// TIA Portal V19 export
TYPE "LUC_typeMonitoring"
TITLE = LUC_typeStateModeManagerMonitoring
// Module related monitoring information
// stored: Access Published
   STRUCT
      unitModeCurrent { ExternalWritable := 'False'} : DInt;   // Current unit mode
      unitModeRequested { ExternalWritable := 'False'} : Bool;   // Requested unit mode change
      unitModeChangeInProcess { ExternalWritable := 'False'} : Bool;   // Unit mode change in process
      stateCurrent { ExternalWritable := 'False'} : DInt;   // Current state
      stateRequested { ExternalWritable := 'False'} : DInt;   // Requested state
      stateChangeInProcess { ExternalWritable := 'False'} : Bool;   // State change in process
      curDisabledStates { ExternalWritable := 'False'} : DWord;   // Disabled states in current unit mode
      curHoldCmdCfg { ExternalWritable := 'False'} : DWord;   // Bit locations within the DWORD represent State numbers. A value of 1 in a bit location indicates that the Hold control command is taken into account in the corresponding state
      curCompleteCmdCfg { ExternalWritable := 'False'} : DWord;   // Bit locations within the DWORD represent State numbers. A value of 1 in a bit location indicates that the Complete control command is taken into account in the corresponding state
      curEnabledModes { ExternalWritable := 'False'} : DWord;   // Bit locations within the DWORD represent Mode numbers. A value of 1 in a bit location [0-31] indicates that the corresponding Mode number is enabled. Mode 0 is an Invalid Mode, therefore bit 0 is unused
      allowedUnitModes { ExternalWritable := 'False'} : DWord;   // Bit locations within the DWORD represent Mode numbers. A value of 1 in a bit location [0-31] indicates that a change to the corresponding Mode number is currently possible. Mode 0 is an Invalid Mode, therefore bit 0 is unused
      cntrlCmdNotAllowed { ExternalWritable := 'False'} : Bool;   // Control command is not allowed (output is reset with the next successful CntrlCmd or if input 'CntrlCmd' is set to 0 or if input 'CmdChangeRequest' is set to FALSE)
      localControlEnabled { ExternalWritable := 'False'} : Bool;   // Local control of the unit mode state manager is enabled
      hmiControlEnabled { ExternalWritable := 'False'} : Bool;   // Hmi control of the unit mode state manager is enabled
      remoteControlEnabled { ExternalWritable := 'False'} : Bool;   // Remote control of the unit mode state manager is enabled
   END_STRUCT;
END_TYPE
